ADAPTER ASR2 (* bidirectional Adapter Interface for 2 Events *)
  (* Standard: 61499-1 *)
  (* Version 1.0, 2025-05-27, franz *)
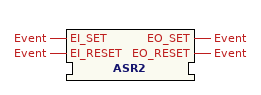
  EVENT_INPUT
    EI_SET; (* Set / Switch on *)
    EI_RESET; (* Reset / Switch off *)
  END_EVENT
  EVENT_OUTPUT
    EO_SET; (* Set / Switch on *)
    EO_RESET; (* Reset / Switch off *)
  END_EVENT
END_ADAPTER
